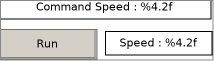
VISUALIZATION ConveyorAuto  // 214x61
VAR_IN_OUT
	bRunConveyor : BOOL;
	fActualSpeed : LREAL;
	fCmdSpeed : LREAL;
END_VAR
    Rectangle (-2,-5 213x24), "Command Speed : %4.2f", text variable: fCmdSpeed
        OnMouseClick: write fCmdSpeed via Edit, min 1, max 2000
    Button (-2,29 99x30), "Run"
        toggle bRunConveyor
    Rectangle (105,31 107x24), "Speed : %4.2f", text variable: fActualSpeed
END_VISUALIZATION

(* stored: Version 1.1.0.1
   Visu ConveyorAuto: Id {742064b2-2ec8-463b-a99c-250e06fc2ce3} *)
